# EPICS alarm handler configuration: mps_database/bareTest/alarms/areas/mpln_sps_mp05.alhConfig
GROUP NULL MPLN:SPS:MP05:1
$ALIAS MPS Link Node 196
$GUIDANCE
LTUH MPS
   Group Name: MPLN:SPS:MP05:1
   Summary PV:  MPLN:SPS:MP05:1:STATSUMY
$END
CHANNEL  MPLN:SPS:MP05:1    MPLN:SPS:MP05:1:MPS_EN_RBV		-----
CHANNEL  MPLN:SPS:MP05:1    MPLN:SPS:MP05:1:LC1_MODE_RBV		-----
